FUNCTION F_Log : BOOL
VAR_INPUT
	fbMessage:			REFERENCE TO FB_Message;
END_VAR
VAR
	sMessage:			STRING(255):= 'Logger null | ';
	ir: INT;
END_VAR

IF fbMessage.bRaised THEN
	;
ELSE
	fbMessage.bRaised:= TRUE;
	sMessage:= CONCAT(sMessage, fbMessage.sSource);
	IF fbMessage.sType <> '' THEN
		sMessage:= CONCAT(sMessage, ' - ');
		sMessage:= CONCAT(sMessage, fbMessage.sType);		
	END_IF
	sMessage:= CONCAT(sMessage, ' |');
	IF fbMessage.nID <> 0 THEN
		sMessage:= CONCAT(sMessage, ' ID: ');
		sMessage:= CONCAT(sMessage, UDINT_TO_STRING(fbMessage.nID));		
		sMessage:= CONCAT(sMessage, ' ');
	END_IF
	sMessage:= CONCAT(sMessage, TO_STRING(fbMessage.eLogLevel));
	sMessage:= CONCAT(sMessage, ': ');
	sMessage:= CONCAT(sMessage, fbMessage.sDefault);
	
	CASE fbMessage.eLogLevel OF
		
		E_LogLevel.Verbose, E_LogLevel.Info:
			ADSLOGSTR(ADSLOG_MSGTYPE_HINT, '%s', sMessage);
			
		E_LogLevel.Warning:
			ADSLOGSTR(ADSLOG_MSGTYPE_WARN, '%s', sMessage);
	
		E_LogLevel.Error, E_LogLevel.Critical:
			ADSLOGSTR(ADSLOG_MSGTYPE_ERROR, '%s', sMessage);
	
	END_CASE

END_IF

END_FUNCTION

(* stored: Version 1.1.0.1
   POU F_Log: Id {3d8b8d8d-2aeb-485f-a382-76004536aaec}, SpecialFunc None *)
